(* CODESYS project PLC_PRG.xml

Project tree, tasks and I/O mapping:
  program PLC_PRG [ST]
*)

// PLC_PRG
PROGRAM PLC_PRG
VAR
END_VAR

END_PROGRAM
